FUNCTION_BLOCK FB_Coating_States EXTENDS FB_PositionStateBase_WithPMPS
VAR_INPUT
    {attribute 'pytmc' := '
      pv: SET
      io: io
    '}
    enumSet : ENUM_Coating_States;
    
    stCoating1 : DUT_PositionState;
    stCoating2 : DUT_PositionState;

    sPmpsDeviceName: STRING;
    sTransitionKey: STRING;
END_VAR
VAR_OUTPUT
	{attribute 'pytmc' := '
      pv: GET;
      io: i;
    '}
    enumGet : ENUM_Coating_States;
  END_VAR
VAR
	bCoatingInit : BOOL;
END_VAR

if NOT bCoatingInit THEN
    bCoatingInit := TRUE;
	
    arrStates[1] := stCoating1;
	arrStates[2] := stCoating2;
END_IF

setState := enumSet;
Exec();
enumGet := getState;
enumSet := setState;

END_FUNCTION_BLOCK

(* stored: Version 1.1.0.1, ProductVersion 3.1.4022.18
   POU FB_Coating_States: Id {dd48993e-b2f6-4df2-ba10-a9b50dee131a}, SpecialFunc None *)
